FUNCTION_BLOCK SC_FirstFloor EXTENDS FB_Chain
VAR_INPUT
	bExecute : BOOL;
	bIncomingPallet : BOOL;
	bPostPalletizerRequestGranted : BOOL;
END_VAR
VAR_OUTPUT
	bPlateOpen : BOOL;
	bPalletizerRequest : BOOL;
	bSentToPostPalletizer : BOOL;
	bPostPalletizerDeliveryRequest : BOOL;
END_VAR
VAR
	fbPallChainConveyor : PalletizerConveyor;
	fbPallElevator : PalletizerElevator;
	fbPlateCyl : Cylinder;
	fbPlateLimitSen : Sensor;
	fbElevatorFrontLimit : Sensor;
	fbElevatorBackLimit : Sensor;
END_VAR

SUPER^();
bPlateOpen := fbPlateCyl.bExtended;
fbPallChainConveyor();
fbPallElevator();
fbPlateCyl();
fbPlateLimitSen();

METHOD PROTECTED   Busy : BOOL
VAR_INPUT
END_VAR

		
fbStepWorkerBusy();
CASE fbStepWorkerBusy.uiStep OF
	
	0: 
		fbPallChainConveyor.On();
		fbStepWorkerBusy
			.mAddCondition(itfStepCondition := fbElevatorBackLimit.getSignal)
			.mAddCondition(itfStepCOndition := fbElevatorFrontLimit.getSignal)
			.mNextStep(10);
			
	10: 
	
		fbPallChainConveyor.Off();
		bPalletizerRequest := FALSE;
		IF rChainController
			.releaseCheck(THIS^)
			.releaseFromChain(sChainReleasing := 'scSecondFloor', THIS^)
			.releaseResult(THIS^) 
		THEN
			fbStepWorkerBusy.mNextStep(20);
		END_IF

	20:
	
		fbPallElevator.MoveUp();
		fbStepWorkerBusy
			.mSetTimer(T#1S)
			.mNextStep(30);
			
	30:
	
		IF NOT fbPallElevator.isMoving
		THEN
			fbStepWorkerBusy
				.mSetTimer(tTime := T#2S)
				.mNextStep(40);
		END_IF
		
	40:
	
		fbPlateCyl.Extend();
		fbStepWorkerBusy
			.mSetTimer(T#2S)
			.mNextStep(45);
	
	45:	
		rChainController.releaseForChain('scSecondFloor', THIS^);	
		fbPallElevator.MoveDown();		
		fbStepWorkerBusy
			.mSetTimer(T#2S)
			.mNextStep(50);
	50:
	
		IF NOT fbPallElevator.isMoving
		THEN
			rChainController.releaseForChain('scPostPalletizer', THIS^);
			fbStepWorkerBusy.mNextStep(60);
		END_IF
	
		
	60:
	
		fbPlateCyl.Retract();
		fbStepWorkerBusy.mNextStep(100);
	
	100:
	
		IF rChainController
			.releaseCheck(THIS^)
			.releaseFromChain(sChainReleasing := 'scPostPalletizer', THIS^)
			.releaseResult(THIS^) 
		THEN

			fbPallChainConveyor.On();
			fbStepWorkerBusy.mNextStep(105);
			
		END_IF

	105:
		fbStepWorkerBusy
				.mSetTimer(T#2s)
				.mNextStep(110);
	110:		
		
		IF NOT fbElevatorBackLimit.bSignal
			AND NOT fbElevatorFrontLimit.bSignal
		THEN
		
			Done();
			fbPallChainConveyor.Off();
			fbStepWorkerBusy.mNextStep(0);
		END_IF

END_CASE
END_METHOD

METHOD PROTECTED  Error : BOOL
VAR_INPUT
END_VAR
END_METHOD

METHOD PROTECTED  Idle : BOOL
VAR_INPUT
END_VAR
END_METHOD

METHOD PROTECTED  Init : BOOL
VAR_INPUT
END_VAR
Start();
END_METHOD

METHOD PROTECTED  Prepare : BOOL
VAR_INPUT
END_VAR
END_METHOD

METHOD PROTECTED  Ready : BOOL
VAR_INPUT
END_VAR

fbStepWorkerReady();
CASE fbStepWorkerReady.uiStep OF
	
	0: 
	
		IF bExecute THEN
			fbStepWorkerReady.mNextStep(10);
		END_IF
		
	10:

		IF NOT fbElevatorFrontLimit.bSignal
			AND NOT fbElevatorBackLimit.bSignal 
		THEN
			bPalletizerRequest := TRUE;
			fbStepWorkerReady.mNextStep(20);
		END_IF
		
	20:
	
		IF bIncomingPallet
		THEN
			fbStepWorkerReady.mNextStep(0);
			Execute();
		END_IF
		
		
END_CASE
END_METHOD

METHOD PROTECTED  Waiting : BOOL
VAR_INPUT
END_VAR
END_METHOD

END_FUNCTION_BLOCK

(* stored: Version 1.1.0.1, ProductVersion 3.1.4024.2
   POU SC_FirstFloor: Id {332726e3-5481-4e2e-85da-27a3a0cd6ff5}, SpecialFunc None
   Method Busy: Id {5fa6aa42-4801-49f4-9f34-075144b33abe}
   Method Error: Id {67dff972-c9e3-421a-9a8a-86234dbb4529}
   Method Idle: Id {0677231a-bfef-4e8d-80f3-5dd0ee6fd95f}
   Method Init: Id {38988075-7506-49ba-b805-efd39e0aa16a}
   Method Prepare: Id {3c8ccc3f-bea7-4d3c-bbcb-40128bc17866}
   Method Ready: Id {7b81569e-0a88-45f1-b024-7895dd9ea9aa}
   Method Waiting: Id {4f6c61b2-bd27-455c-8184-81eaa16069d7} *)
